// TIA Portal V18 export
DATA_BLOCK "Data_block_2"   // DB3
{ S7_Optimized_Access := 'TRUE' }
VERSION : 0.1
// stored: AutoNumber true, IsOnlyStoredInLoadMemory false, IsRetainMemResEnabled false, IsWriteProtectedInAS false, MemoryReserve 100
   VAR
      ar : Array[0..1000] of Time_Of_Day;
   END_VAR
BEGIN
END_DATA_BLOCK
